// TIA Portal V20 export
FUNCTION_BLOCK "LER_DWordToDInt"   // FB99, LAD
// stored: Access Published, MemoryReserve 100, SetENOAutomatically false
   VAR_INPUT
      Input1 : DWord;
      Input2 : DWord;
      Input3 : DWord;
      Input4 : DWord;
      Input5 : DWord;
      Input6 : DWord;
      Input7 : DWord;
      Input8 : DWord;
      Input9 : DWord;
      Input10 : DWord;
   END_VAR
   VAR_OUTPUT
      Output1 : DInt;
      Output2 : DInt;
      Output3 : DInt;
      Output4 : DInt;
      Output5 : DInt;
      Output6 : DInt;
      Output7 : DInt;
      Output8 : DInt;
      Output9 : DInt;
      Output10 : DInt;
   END_VAR
BEGIN

REGION Network 1
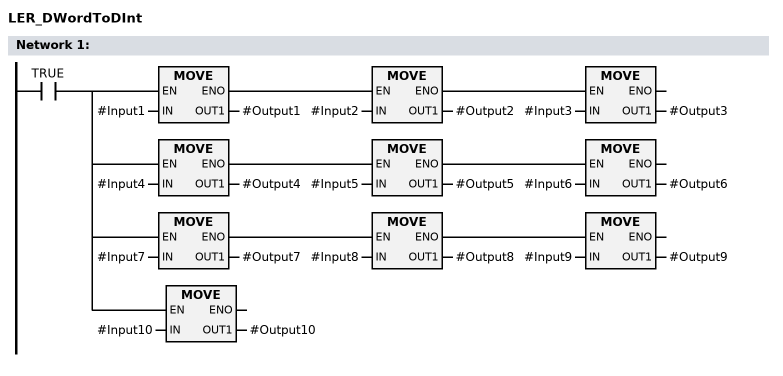
   RUNG wire#powerrail
      Contact( TRUE )
      wire#w1
      Move(in := #Input1, out1 => #Output1)
      Move(in := #Input2, out1 => #Output2)
      Move(in := #Input3, out1 => #Output3)
   END_RUNG
   RUNG wire#w1
      Move(in := #Input4, out1 => #Output4)
      Move(in := #Input5, out1 => #Output5)
      Move(in := #Input6, out1 => #Output6)
   END_RUNG
   RUNG wire#w1
      Move(in := #Input7, out1 => #Output7)
      Move(in := #Input8, out1 => #Output8)
      Move(in := #Input9, out1 => #Output9)
   END_RUNG
   RUNG wire#w1
      Move(in := #Input10, out1 => #Output10)
   END_RUNG
   // the same network as SCL:
   IF TRUE THEN
       #Output1 := #Input1;
       #Output2 := #Input2;
       #Output3 := #Input3;
       #Output4 := #Input4;
       #Output5 := #Input5;
       #Output6 := #Input6;
       #Output7 := #Input7;
       #Output8 := #Input8;
       #Output9 := #Input9;
       #Output10 := #Input10;
   END_IF;
END_REGION
END_FUNCTION_BLOCK
